FUNCTION_BLOCK ReadAssigment
VAR_INPUT
	assigment : Auftrag;
END_VAR
VAR_OUTPUT
	lastPointsToPickup : ARRAY[0..2] OF RobotPoseSimple;		//Weg zum Abholort (letzte Punkte)
	pointsFromSlotToReader : ARRAY[0..2] OF RobotPoseSimple;	//Weg vom Abholort zur Abmeldung 
	lastPointsToStorage : ARRAY[0..2] OF RobotPoseSimple;		//Weg zum Ablageort (letzte Punkte)
	pointsFromReaderToSlot : ARRAY[0..2] OF RobotPoseSimple;	//Weg vom Abmelden zur Ablage
	lastNodePickUp, lastNodeStorage : RobotPoseSimple;			//letzter Knoten vor Abholung/Ablage
END_VAR
VAR
	pickupLocation, readerCheckOut, readerCheckIn, storageLocation : RobotPoseSimple;	//Koordinaten der Stationen
	Failed : BOOL := FALSE;
END_VAR

//FB zur Verarbeitung der Daten, die aus dem Auftrag kommen
//es werden Wegpunkte zum Anhängen an die Wegpunktliste und auch Wegpunktlisten zur An- und Abmeldung am RFID Reader generiert


//RFID Leser für Abmeldung
IF assigment.AbholStation = 1 THEN
	IF assigment.AbholTasche = 1 THEN
		//RFID links anfahren
		lastNodePickUp := ToRobotPoseSimple(x := 600, y := 3000, theta := -1); //600?
		pickupLocation := ToRobotPoseSimple(x := 898, y := 2838, theta := 0);
		readerCheckOut := ToRobotPoseSimple(x := 886, y := 2936, theta := 0);
	ELSIF assigment.AbholTasche = 2 THEN
		//RFID links anfahren
		lastNodePickUp := ToRobotPoseSimple(x := 600, y := 2600, theta := -1); //600?
		pickupLocation := ToRobotPoseSimple(x := 898, y := 2739, theta := 0);
		readerCheckOut := ToRobotPoseSimple(x := 886, y := 2936, theta := 0);
	ELSIF assigment.AbholTasche = 3 THEN
		//RFID rechts anfahren
		lastNodePickUp := ToRobotPoseSimple(x := 1400, y := 3000, theta := -1);
		pickupLocation := ToRobotPoseSimple(x := 1311, y := 2835, theta := 0);
		readerCheckOut := ToRobotPoseSimple(x := 1303, y := 2935, theta := 0);	
	ELSIF assigment.AbholTasche = 4 THEN
		//RFID rechts anfahren	
		lastNodePickUp := ToRobotPoseSimple(x := 1400, y := 2600, theta := -1);
		pickupLocation := ToRobotPoseSimple(x := 1310, y := 2736, theta := 0);
		readerCheckOut := ToRobotPoseSimple(x := 1303, y := 2935, theta := 0);			
	ELSE
		//Fehler
		Failed := TRUE;
	END_IF
ELSIF assigment.AbholStation = 2 THEN
	IF assigment.AbholTasche = 1 THEN
		//RFID links anfahren
		lastNodePickUp := ToRobotPoseSimple(x := 1800, y := 3000, theta := -1);
		pickupLocation := ToRobotPoseSimple(x := 2099, y := 2829, theta := 0);
		readerCheckOut := ToRobotPoseSimple(x := 2088, y := 2931, theta := 0);	
	ELSIF assigment.AbholTasche = 2 THEN
		//RFID links anfahren
		lastNodePickUp := ToRobotPoseSimple(x := 1800, y := 2600, theta := -1);
		pickupLocation := ToRobotPoseSimple(x := 2099, y := 2731, theta := 0);
		readerCheckOut := ToRobotPoseSimple(x := 2088, y := 2931, theta := 0);	
	ELSIF assigment.AbholTasche = 3 THEN
		//RFID rechts anfahren
		lastNodePickUp := ToRobotPoseSimple(x := 2600, y := 3000, theta := -1);
		pickupLocation := ToRobotPoseSimple(x := 2438, y := 2833, theta := 0);
		readerCheckOut := ToRobotPoseSimple(x := 2433, y := 2937, theta := 0);		
	ELSIF assigment.AbholTasche = 4 THEN
		//RFID rechts anfahren
		lastNodePickUp := ToRobotPoseSimple(x := 2600, y := 2600, theta := -1);
		pickupLocation := ToRobotPoseSimple(x := 2437, y := 2732, theta := 0);
		readerCheckOut := ToRobotPoseSimple(x := 2433, y := 2937, theta := 0);			
	ELSE
		//Fehler
		Failed := TRUE;
	END_IF
ELSIF assigment.AbholStation = 3 THEN
	IF assigment.AbholTasche = 1 THEN
		//RFID links anfahren
		lastNodePickUp := ToRobotPoseSimple(x := 3000, y := 3000, theta := -1);
		pickupLocation := ToRobotPoseSimple(x := 3229, y := 2837, theta := 0);
		readerCheckOut := ToRobotPoseSimple(x := 3235, y := 2941, theta := 0);
	ELSIF assigment.AbholTasche = 2 THEN
		//RFID links anfahren
		lastNodePickUp := ToRobotPoseSimple(x := 3000, y := 2600, theta := -1);
		pickupLocation := ToRobotPoseSimple(x := 3228, y := 2732, theta := 0);
		readerCheckOut := ToRobotPoseSimple(x := 3235, y := 2941, theta := 0);
	ELSIF assigment.AbholTasche = 3 THEN
		//RFID rechts anfahren
		lastNodePickUp := ToRobotPoseSimple(x := 3800, y := 3000, theta := -1);
		pickupLocation := ToRobotPoseSimple(x := 3653, y := 2840, theta := 0);
		readerCheckOut := ToRobotPoseSimple(x := 3658, y := 2939, theta := 0);	
	ELSIF assigment.AbholTasche = 4 THEN
		//RFID rechts anfahren
		lastNodePickUp := ToRobotPoseSimple(x := 3800, y := 2600, theta := -1);
		pickupLocation := ToRobotPoseSimple(x := 3650, y := 2732, theta := 0);
		readerCheckOut := ToRobotPoseSimple(x := 3658, y := 2939, theta := 0);			
	ELSE
		//Fehler
		Failed := TRUE;
	END_IF
ELSIF assigment.AbholStation = 4 THEN
	IF assigment.AbholTasche = 1 THEN
		//RFID links anfahren
		lastNodePickUp := ToRobotPoseSimple(x := 4200, y := 3000, theta := -1);
		pickupLocation := ToRobotPoseSimple(x := 4450, y := 2838, theta := 0);
		readerCheckOut := ToRobotPoseSimple(x := 4449, y := 2937, theta := 0);
	ELSIF assigment.AbholTasche = 2 THEN
		//RFID links anfahren
		lastNodePickUp := ToRobotPoseSimple(x := 4200, y := 2600, theta := -1);
		pickupLocation := ToRobotPoseSimple(x := 4449, y := 2732, theta := 0);
		readerCheckOut := ToRobotPoseSimple(x := 4449, y := 2937, theta := 0);
	ELSIF assigment.AbholTasche = 3 THEN
		//RFID rechts anfahren
		lastNodePickUp := ToRobotPoseSimple(x := 5000, y := 3000, theta := -1);
		pickupLocation := ToRobotPoseSimple(x := 4879, y := 2844, theta := 0);
		readerCheckOut := ToRobotPoseSimple(x := 4893, y := 2946, theta := 0);	
	ELSIF assigment.AbholTasche = 4 THEN
		//RFID rechts anfahren
		lastNodePickUp := ToRobotPoseSimple(x := 5000, y := 2600, theta := -1);
		pickupLocation := ToRobotPoseSimple(x := 4893, y := 2741, theta := 0);
		readerCheckOut := ToRobotPoseSimple(x := 4893, y := 2946, theta := 0);			
	ELSE
		//Fehler
		Failed := TRUE;
	END_IF
ELSE
	//Fehler
	Failed := TRUE;		
END_IF


//Auswählen RFID Leser für Anmeldung
IF assigment.AblageStation = 1 THEN
	IF assigment.AblageTasche = 1 THEN
		//RFID links anfahren
		lastNodeStorage := ToRobotPoseSimple(x := 600, y := 3000, theta := -1); //600?
		storageLocation := ToRobotPoseSimple(x := 898, y := 2838, theta := 0);
		readerCheckIn := ToRobotPoseSimple(x := 886, y := 2936, theta := 0);
	ELSIF assigment.AblageTasche = 2 THEN
		//RFID links anfahren
		lastNodePickUp := ToRobotPoseSimple(x := 600, y := 2600, theta := -1); //600?
		pickupLocation := ToRobotPoseSimple(x := 898, y := 2739, theta := 0);
		readerCheckOut := ToRobotPoseSimple(x := 886, y := 2936, theta := 0);
	ELSIF assigment.AblageTasche = 3 THEN
		//RFID rechts anfahren	
		lastNodePickUp := ToRobotPoseSimple(x := 1400, y := 3000, theta := -1);
		pickupLocation := ToRobotPoseSimple(x := 1311, y := 2835, theta := 0);
		readerCheckOut := ToRobotPoseSimple(x := 1303, y := 2935, theta := 0);	
	ELSIF assigment.AblageTasche = 4 THEN
		//RFID rechts anfahren	
		lastNodePickUp := ToRobotPoseSimple(x := 1400, y := 2600, theta := -1);
		pickupLocation := ToRobotPoseSimple(x := 1310, y := 2736, theta := 0);
		readerCheckOut := ToRobotPoseSimple(x := 1303, y := 2935, theta := 0);		
	ELSE
		//Fehler
		Failed := TRUE;
	END_IF
ELSIF assigment.AblageStation = 2 THEN
	IF assigment.AblageTasche = 1 THEN
		//RFID links anfahren
		lastNodePickUp := ToRobotPoseSimple(x := 1800, y := 3000, theta := -1);
		pickupLocation := ToRobotPoseSimple(x := 2099, y := 2829, theta := 0);
		readerCheckOut := ToRobotPoseSimple(x := 2088, y := 2931, theta := 0);	
	ELSIF assigment.AblageTasche = 2 THEN
		//RFID links anfahren
		lastNodePickUp := ToRobotPoseSimple(x := 1800, y := 2600, theta := -1);
		pickupLocation := ToRobotPoseSimple(x := 2099, y := 2731, theta := 0);
		readerCheckOut := ToRobotPoseSimple(x := 2088, y := 2931, theta := 0);
	ELSIF assigment.AblageTasche = 3 THEN
		//RFID rechts anfahren	
		lastNodePickUp := ToRobotPoseSimple(x := 2600, y := 3000, theta := -1);
		pickupLocation := ToRobotPoseSimple(x := 2438, y := 2833, theta := 0);
		readerCheckOut := ToRobotPoseSimple(x := 2433, y := 2937, theta := 0);	
	ELSIF assigment.AblageTasche = 4 THEN
		//RFID rechts anfahren	
		lastNodePickUp := ToRobotPoseSimple(x := 2600, y := 2600, theta := -1);
		pickupLocation := ToRobotPoseSimple(x := 2437, y := 2732, theta := 0);
		readerCheckOut := ToRobotPoseSimple(x := 2433, y := 2937, theta := 0);			
	ELSE
		//Fehler
		Failed := TRUE;
	END_IF
ELSIF assigment.AblageStation = 3 THEN
	IF assigment.AblageTasche = 1 THEN
		//RFID links anfahren
		lastNodePickUp := ToRobotPoseSimple(x := 3000, y := 3000, theta := -1);
		pickupLocation := ToRobotPoseSimple(x := 3229, y := 2837, theta := 0);
		readerCheckOut := ToRobotPoseSimple(x := 3235, y := 2941, theta := 0);
	ELSIF assigment.AblageTasche = 2 THEN
		//RFID links anfahren
		lastNodePickUp := ToRobotPoseSimple(x := 3000, y := 2600, theta := -1);
		pickupLocation := ToRobotPoseSimple(x := 3228, y := 2732, theta := 0);
		readerCheckOut := ToRobotPoseSimple(x := 3235, y := 2941, theta := 0);
	ELSIF assigment.AblageTasche = 3 THEN
		//RFID rechts anfahren
		lastNodePickUp := ToRobotPoseSimple(x := 3800, y := 3000, theta := -1);
		pickupLocation := ToRobotPoseSimple(x := 3653, y := 2840, theta := 0);
		readerCheckOut := ToRobotPoseSimple(x := 3658, y := 2939, theta := 0);		
	ELSIF assigment.AblageTasche = 4 THEN
		//RFID rechts anfahren	
		lastNodePickUp := ToRobotPoseSimple(x := 3800, y := 2600, theta := -1);
		pickupLocation := ToRobotPoseSimple(x := 3650, y := 2732, theta := 0);
		readerCheckOut := ToRobotPoseSimple(x := 3658, y := 2939, theta := 0);		
	ELSE
		//Fehler
		Failed := TRUE;
	END_IF
ELSIF assigment.AblageStation = 4 THEN
	IF assigment.AblageTasche = 1 THEN
		//RFID links anfahren
		lastNodePickUp := ToRobotPoseSimple(x := 4200, y := 3000, theta := -1);
		pickupLocation := ToRobotPoseSimple(x := 4450, y := 2838, theta := 0);
		readerCheckOut := ToRobotPoseSimple(x := 4449, y := 2937, theta := 0);
	ELSIF assigment.AblageTasche = 2 THEN
		//RFID links anfahren
		lastNodePickUp := ToRobotPoseSimple(x := 4200, y := 2600, theta := -1);
		pickupLocation := ToRobotPoseSimple(x := 4449, y := 2732, theta := 0);
		readerCheckOut := ToRobotPoseSimple(x := 4449, y := 2937, theta := 0);
	ELSIF assigment.AblageTasche = 3 THEN
		//RFID rechts anfahren	
		lastNodePickUp := ToRobotPoseSimple(x := 5000, y := 3000, theta := -1);
		pickupLocation := ToRobotPoseSimple(x := 4879, y := 2844, theta := 0);
		readerCheckOut := ToRobotPoseSimple(x := 4893, y := 2946, theta := 0);
	ELSIF assigment.AblageTasche = 4 THEN
		//RFID rechts anfahren	
		lastNodePickUp := ToRobotPoseSimple(x := 5000, y := 2600, theta := -1);
		pickupLocation := ToRobotPoseSimple(x := 4893, y := 2741, theta := 0);
		readerCheckOut := ToRobotPoseSimple(x := 4893, y := 2946, theta := 0);		
	ELSE
		//Fehler
		Failed := TRUE;
	END_IF
ELSE
	//Fehler
	Failed := TRUE;		
END_IF


//Abholort (3 Punkte) an Wegpunktliste anfügen
//lastPointsToPickup[0] := lastNodePickUp;
lastPointsToPickup[1] := ToRobotPoseSimple(x := lastNodePickUp.x, y := pickupLocation.y, theta := pickupLocation.theta);
lastPointsToPickup[2] := pickupLocation;

//erstellen 3 Wegpunkte für fahren von Tasche zu RFID Leser
pointsFromSlotToReader[0] := ToRobotPoseSimple(x := lastNodePickUp.x, y := pickupLocation.y, theta := pickupLocation.theta);
pointsFromSlotToReader[1] := ToRobotPoseSimple(x := lastNodePickUp.x, y := readerCheckOut.y, theta := readerCheckOut.theta);
pointsFromSlotToReader[2] := readerCheckOut;

//Ablageort (3 Punkte) an Wegpunktliste anfügen (Ankunft Reader)
//lastPointsToStorage[0] := lastNodeStorage;
lastPointsToStorage[1] := ToRobotPoseSimple(x := lastNodeStorage.x, y := readerCheckIn.y, theta := readerCheckIn.theta);
lastPointsToStorage[2] := readerCheckIn;

//3 Wegpunkte von RFID Leser zu Ablageort
pointsFromReaderToSlot[0] := ToRobotPoseSimple(x := lastNodeStorage.x, y := readerCheckIn.y, theta := readerCheckIn.theta);
pointsFromReaderToSlot[1] := ToRobotPoseSimple(x := lastNodeStorage.x, y := storageLocation.y, theta := storageLocation.theta);
pointsFromReaderToSlot[2] := storageLocation;

END_FUNCTION_BLOCK

(* stored: Version 1.1.0.1, ProductVersion 3.1.4024.11
   POU ReadAssigment: Id {be20b526-cbde-4de4-80a7-e4ae669afa53}, SpecialFunc None *)
